# EPICS alarm handler configuration: mps_database/bareTest/alarms/areas/mpln_dog_mp01.alhConfig
GROUP NULL MPLN:DOG:MP01:1
$ALIAS MPS Link Node 72
$GUIDANCE
LTUH MPS
   Group Name: MPLN:DOG:MP01:1
   Summary PV:  MPLN:DOG:MP01:1:STATSUMY
$END
CHANNEL  MPLN:DOG:MP01:1    MPLN:DOG:MP01:1:MPS_EN_RBV		-----
CHANNEL  MPLN:DOG:MP01:1    MPLN:DOG:MP01:1:LC1_MODE_RBV		-----
